// TwinCAT 3 PLC project Practice_4
// ProgramVersion: 3.1.4024.0
// libraries:
//   Tc2_Standard, * (Beckhoff Automation GmbH)
//   Tc2_System, * (Beckhoff Automation GmbH)
//   Tc3_Module, * (Beckhoff Automation GmbH)
// project tree:
//   DUTs/ ST_Device.TcDUT
//   / PlcTask.TcTTO
//   POUs/ MAIN.TcPOU
// (motion and I/O tree: see PLC project practice_1)
// real-time tasks:
//   TASK PlcTask: cycle T#10ms, priority 20, ADS port 350
//   TASK PlcTask1: cycle T#10ms, priority 21, ADS port 351
//   TASK PlcTask2: cycle T#10ms, priority 22, ADS port 352
//   TASK PlcTask3: cycle T#10ms, priority 23, ADS port 353

CONFIGURATION Practice_4
    RESOURCE PLC ON TwinCAT3
        TASK PlcTask(INTERVAL := T#10ms, PRIORITY := 23);
        PROGRAM MAIN WITH PlcTask : MAIN;
    END_RESOURCE
END_CONFIGURATION

// ---- DUTs/ST_Device.TcDUT
TYPE ST_Device :
STRUCT
	sDeviceName : STRING;
	nDeviceValue : INT;
END_STRUCT
END_TYPE

// ---- POUs/MAIN.TcPOU
PROGRAM MAIN
VAR
	stDevice1 : ST_Device := (sDeviceName := 'Poco x6', nDeviceValue := 10000);
	stDevice2 : ST_Device := (sDeviceName := 'Samsung s23', nDeviceValue := 30000);
	bToggle : BOOL;
	bNum1 : INT;
END_VAR

END_PROGRAM
